% RSLogix 500 project LINCEBOT.RSS, saved by version 10.00.00.00 %
PROJECT "LINCEBOT"    % processor: MicroLogix 1400 %

PROGRAM FILES
  LAD 2   28 rungs
  LAD 4   10 rungs
  LAD 6   11 rungs
  LAD 8   6 rungs
  LAD 10   5 rungs
  LAD 12   10 rungs
  LAD 14   12 rungs
  LAD 16   4 rungs
  LAD 18   3 rungs
  LAD 20   3 rungs
  LAD 22   3 rungs
  LAD 24   13 rungs
  LAD 26   11 rungs
  LAD 80   9 rungs
  LAD 90   9 rungs
  LAD 100   27 rungs
  LAD 102   6 rungs
  LAD 103   6 rungs
  LAD 104   9 rungs
  LAD 105   8 rungs
  LAD 110   5 rungs
  LAD 111   8 rungs
  LAD 122   2 rungs
  LAD 125   7 rungs
  LAD 126   33 rungs
  LAD 131   2 rungs
  LAD 141   12 rungs
  LAD 150   11 rungs
  LAD 151   11 rungs
  LAD 160   42 rungs
  LAD 161   42 rungs
  LAD 170   10 rungs
  LAD 180   10 rungs
  LAD 70: only END

DATA FILES
  O0 OUTPUT  11 elements
  I1 INPUT  11 elements
  S2 STATUS  66 elements
  B3 BINARY  14 elements
  T4 TIMER  40 elements
  C5 COUNTER  1 elements
  R6 CONTROL  20 elements
  N7 INTEGER  200 elements
  F8 FLOAT  100 elements
  B9   256 elements
  B10   1 elements
  B11   256 elements
  B12   22 elements
  L13   100 elements
  F14   100 elements
  N15   100 elements
  L16   100 elements
  B17   128 elements
  B18   128 elements
  L23   100 elements
  L24   100 elements
  L42   52 elements
  B181   128 elements
  F182   50 elements
  L183   50 elements
  N184   50 elements
  B185   50 elements
  N186   50 elements
  L187   50 elements
  F188   50 elements
  B189   50 elements
  L190   50 elements
  B191   10 elements
  L192   50 elements
  F193   50 elements
  B194   128 elements
  B195   128 elements
  B196   50 elements
  N197   50 elements
  B198   50 elements
  L199   50 elements
  N200   50 elements
  L201   50 elements
  B202   50 elements
  N203   50 elements
  L204   50 elements
  F205   50 elements

LADDER 2
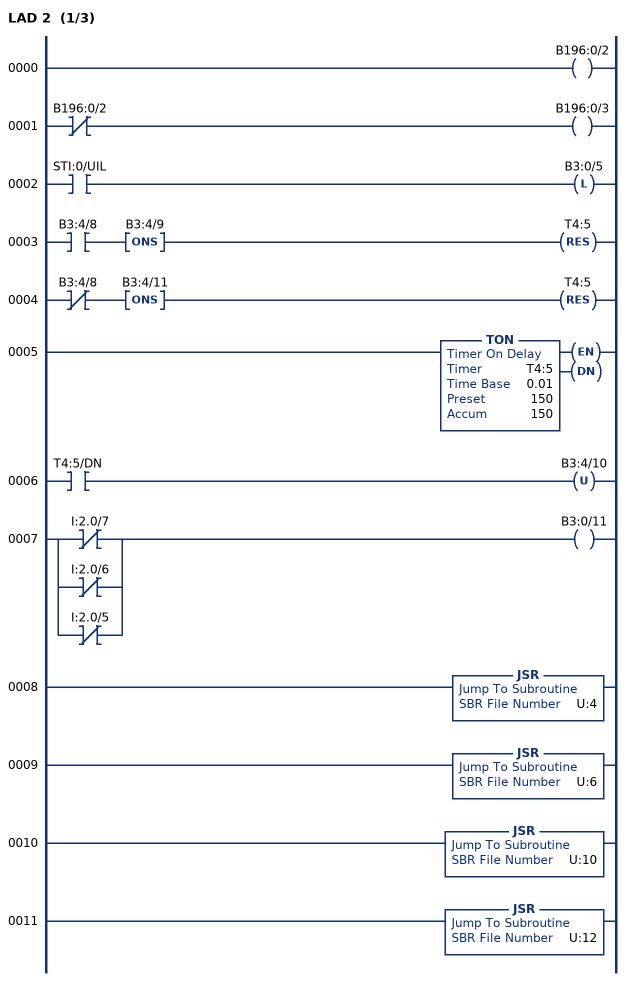
% Rung: 0 %
SOR OTE B196:0/2 EOR
% Rung: 1 %
SOR XIO B196:0/2 OTE B196:0/3 EOR
% Rung: 2 %
SOR XIC STI:0/UIL OTL B3:0/5 EOR
% Rung: 3 %
SOR XIC B3:4/8 ONS B3:4/9 RES T4:5 EOR
% Rung: 4 %
SOR XIO B3:4/8 ONS B3:4/11 RES T4:5 EOR
% Rung: 5 %
SOR TON T4:5 0.01 150 150 EOR
% Rung: 6 %
SOR XIC T4:5/DN OTU B3:4/10 EOR
% Rung: 7 %
SOR BST XIO I:2.0/7 NXB XIO I:2.0/6 NXB XIO I:2.0/5 BND OTE B3:0/11 EOR
% Rung: 8 %
SOR JSR U:4 EOR
% Rung: 9 %
SOR JSR U:6 EOR
% Rung: 10 %
SOR JSR U:10 EOR
% Rung: 11 %
SOR JSR U:12 EOR

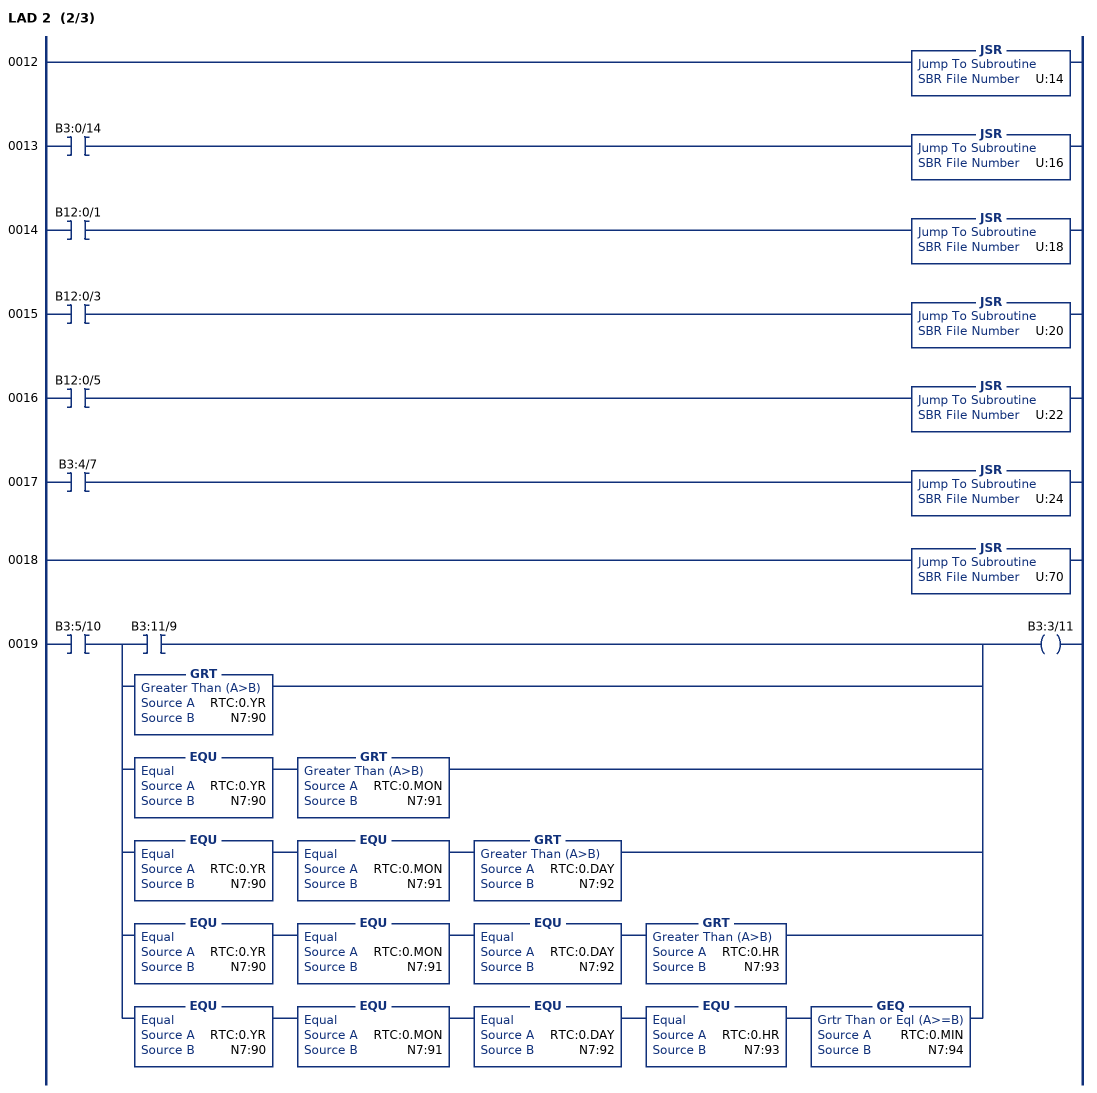
% Rung: 12 %
SOR JSR U:14 EOR
% Rung: 13 %
SOR XIC B3:0/14 JSR U:16 EOR
% Rung: 14 %
SOR XIC B12:0/1 JSR U:18 EOR
% Rung: 15 %
SOR XIC B12:0/3 JSR U:20 EOR
% Rung: 16 %
SOR XIC B12:0/5 JSR U:22 EOR
% Rung: 17 %
SOR XIC B3:4/7 JSR U:24 EOR
% Rung: 18 %
SOR JSR U:70 EOR
% Rung: 19 %
SOR XIC B3:5/10 BST XIC B3:11/9 NXB GRT RTC:0.YR N7:90 NXB EQU RTC:0.YR N7:90 GRT RTC:0.MON N7:91 NXB EQU RTC:0.YR N7:90 EQU RTC:0.MON N7:91 GRT RTC:0.DAY N7:92 NXB EQU RTC:0.YR N7:90 EQU RTC:0.MON N7:91 EQU RTC:0.DAY N7:92 GRT RTC:0.HR N7:93 NXB EQU RTC:0.YR N7:90 EQU RTC:0.MON N7:91 EQU RTC:0.DAY N7:92 EQU RTC:0.HR N7:93 GEQ RTC:0.MIN N7:94 BND OTE B3:3/11 EOR

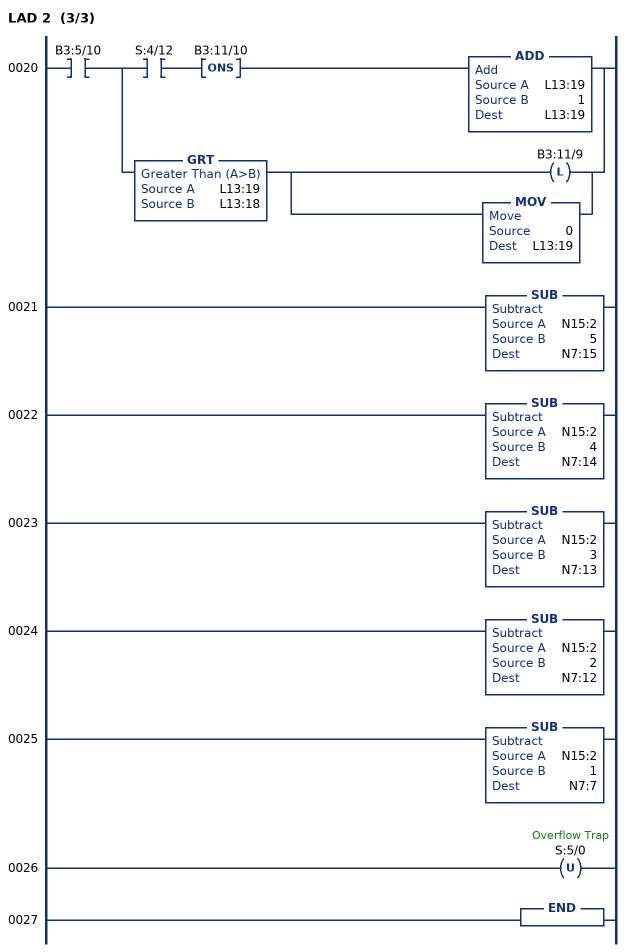
% Rung: 20 %
SOR XIC B3:5/10 BST XIC S:4/12 ONS B3:11/10 ADD L13:19 1 L13:19 NXB GRT L13:19 L13:18 BST OTL B3:11/9 NXB MOV 0 L13:19 BND BND EOR
% Rung: 21 %
SOR SUB N15:2 5 N7:15 EOR
% Rung: 22 %
SOR SUB N15:2 4 N7:14 EOR
% Rung: 23 %
SOR SUB N15:2 3 N7:13 EOR
% Rung: 24 %
SOR SUB N15:2 2 N7:12 EOR
% Rung: 25 %
SOR SUB N15:2 1 N7:7 EOR
% Rung: 26 %
SOR OTU S:5/0 EOR
%   S:5/0  "Overflow Trap" %
% Rung: 27 %
SOR END EOR

LADDER 4
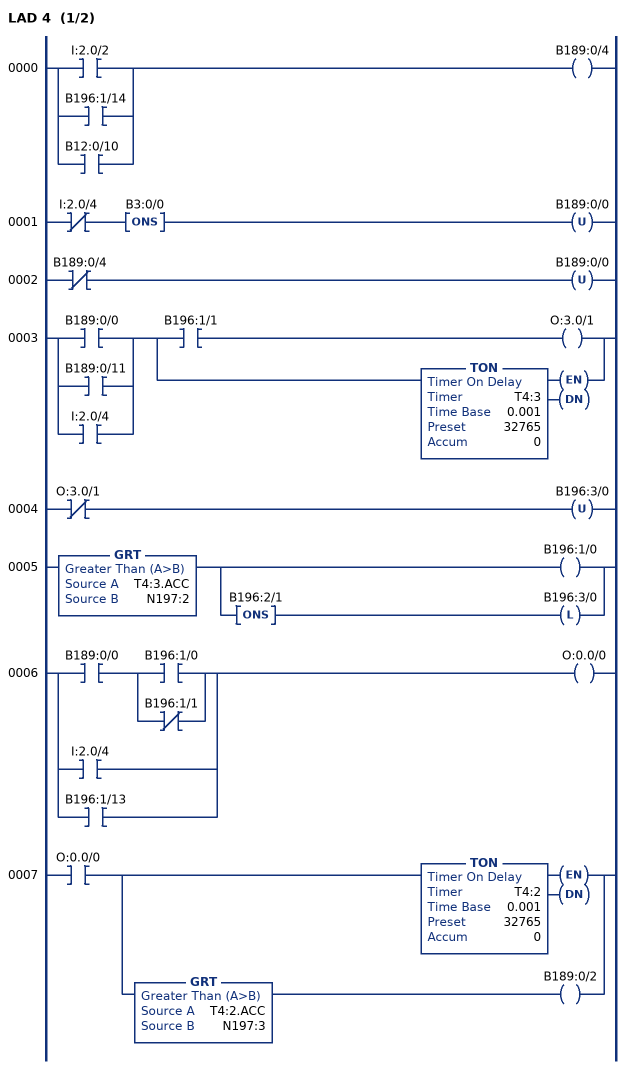
% Rung: 0 %
SOR BST XIC I:2.0/2 NXB XIC B196:1/14 NXB XIC B12:0/10 BND OTE B189:0/4 EOR
% Rung: 1 %
SOR XIO I:2.0/4 ONS B3:0/0 OTU B189:0/0 EOR
% Rung: 2 %
SOR XIO B189:0/4 OTU B189:0/0 EOR
% Rung: 3 %
SOR BST XIC B189:0/0 NXB XIC B189:0/11 NXB XIC I:2.0/4 BND BST XIC B196:1/1 OTE O:3.0/1 NXB TON T4:3 0.001 32765 0 BND EOR
% Rung: 4 %
SOR XIO O:3.0/1 OTU B196:3/0 EOR
% Rung: 5 %
SOR GRT T4:3.ACC N197:2 BST OTE B196:1/0 NXB ONS B196:2/1 OTL B196:3/0 BND EOR
% Rung: 6 %
SOR BST XIC B189:0/0 BST XIC B196:1/0 NXB XIO B196:1/1 BND NXB XIC I:2.0/4 NXB XIC B196:1/13 BND OTE O:0.0/0 EOR
% Rung: 7 %
SOR XIC O:0.0/0 BST TON T4:2 0.001 32765 0 NXB GRT T4:2.ACC N197:3 OTE B189:0/2 BND EOR

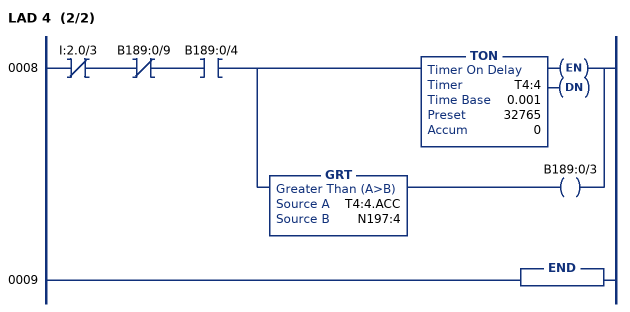
% Rung: 8 %
SOR XIO I:2.0/3 XIO B189:0/9 XIC B189:0/4 BST TON T4:4 0.001 32765 0 NXB GRT T4:4.ACC N197:4 OTE B189:0/3 BND EOR
% Rung: 9 %
SOR END EOR

LADDER 6
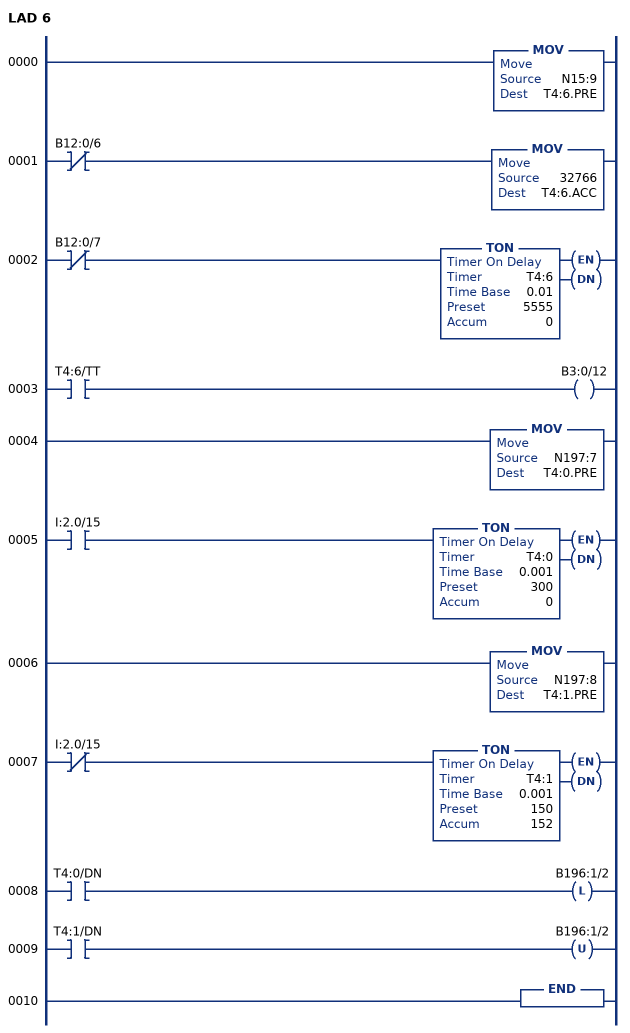
% Rung: 0 %
SOR MOV N15:9 T4:6.PRE EOR
% Rung: 1 %
SOR XIO B12:0/6 MOV 32766 T4:6.ACC EOR
% Rung: 2 %
SOR XIO B12:0/7 TON T4:6 0.01 5555 0 EOR
% Rung: 3 %
SOR XIC T4:6/TT OTE B3:0/12 EOR
% Rung: 4 %
SOR MOV N197:7 T4:0.PRE EOR
% Rung: 5 %
SOR XIC I:2.0/15 TON T4:0 0.001 300 0 EOR
% Rung: 6 %
SOR MOV N197:8 T4:1.PRE EOR
% Rung: 7 %
SOR XIO I:2.0/15 TON T4:1 0.001 150 152 EOR
% Rung: 8 %
SOR XIC T4:0/DN OTL B196:1/2 EOR
% Rung: 9 %
SOR XIC T4:1/DN OTU B196:1/2 EOR
% Rung: 10 %
SOR END EOR

LADDER 8
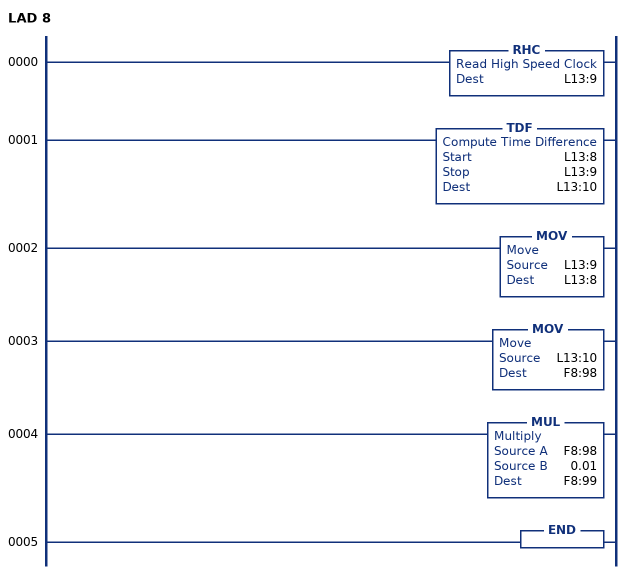
% Rung: 0 %
SOR RHC L13:9 EOR
% Rung: 1 %
SOR TDF L13:8 L13:9 L13:10 EOR
% Rung: 2 %
SOR MOV L13:9 L13:8 EOR
% Rung: 3 %
SOR MOV L13:10 F8:98 EOR
% Rung: 4 %
SOR MUL F8:98 0.01 F8:99 EOR
% Rung: 5 %
SOR END EOR

LADDER 10
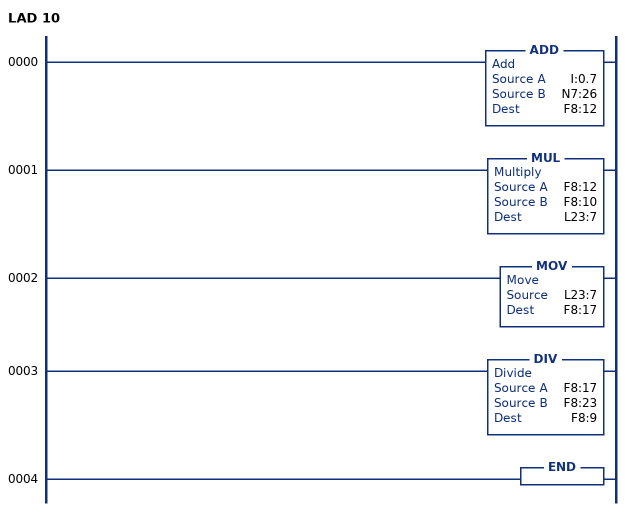
% Rung: 0 %
SOR ADD I:0.7 N7:26 F8:12 EOR
% Rung: 1 %
SOR MUL F8:12 F8:10 L23:7 EOR
% Rung: 2 %
SOR MOV L23:7 F8:17 EOR
% Rung: 3 %
SOR DIV F8:17 F8:23 F8:9 EOR
% Rung: 4 %
SOR END EOR

LADDER 12
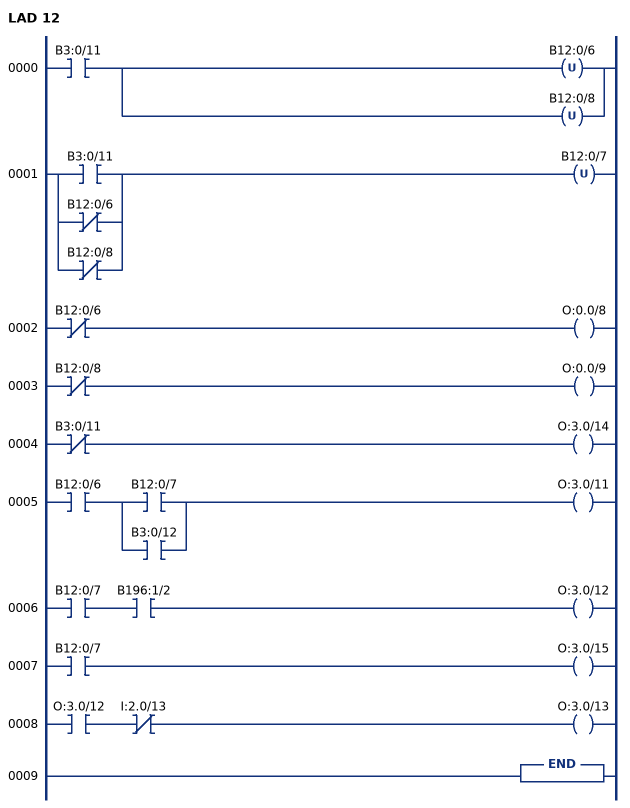
% Rung: 0 %
SOR XIC B3:0/11 BST OTU B12:0/6 NXB OTU B12:0/8 BND EOR
% Rung: 1 %
SOR BST XIC B3:0/11 NXB XIO B12:0/6 NXB XIO B12:0/8 BND OTU B12:0/7 EOR
% Rung: 2 %
SOR XIO B12:0/6 OTE O:0.0/8 EOR
% Rung: 3 %
SOR XIO B12:0/8 OTE O:0.0/9 EOR
% Rung: 4 %
SOR XIO B3:0/11 OTE O:3.0/14 EOR
% Rung: 5 %
SOR XIC B12:0/6 BST XIC B12:0/7 NXB XIC B3:0/12 BND OTE O:3.0/11 EOR
% Rung: 6 %
SOR XIC B12:0/7 XIC B196:1/2 OTE O:3.0/12 EOR
% Rung: 7 %
SOR XIC B12:0/7 OTE O:3.0/15 EOR
% Rung: 8 %
SOR XIC O:3.0/12 XIO I:2.0/13 OTE O:3.0/13 EOR
% Rung: 9 %
SOR END EOR

LADDER 14
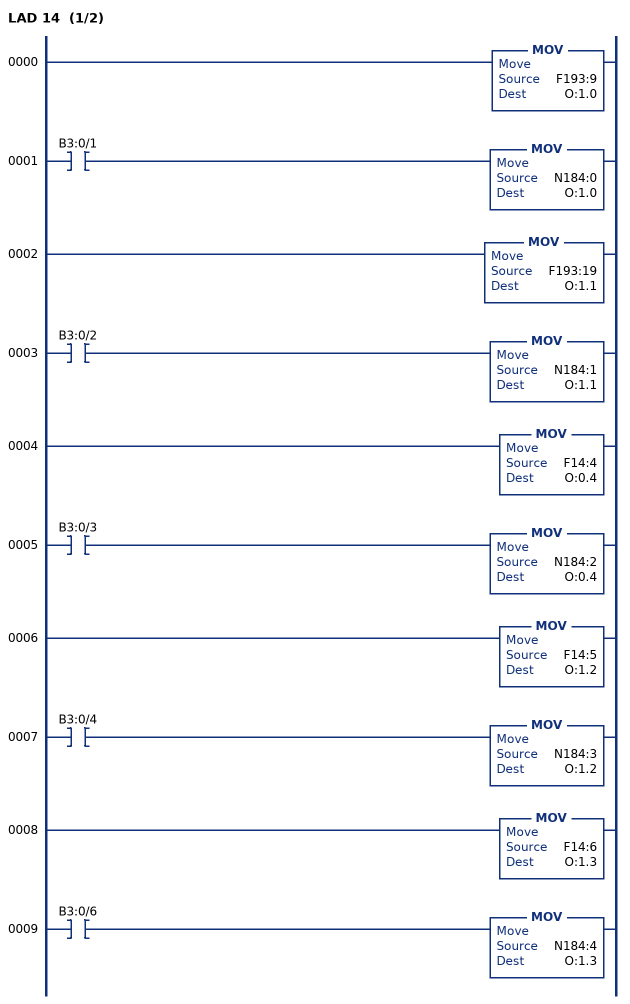
% Rung: 0 %
SOR MOV F193:9 O:1.0 EOR
% Rung: 1 %
SOR XIC B3:0/1 MOV N184:0 O:1.0 EOR
% Rung: 2 %
SOR MOV F193:19 O:1.1 EOR
% Rung: 3 %
SOR XIC B3:0/2 MOV N184:1 O:1.1 EOR
% Rung: 4 %
SOR MOV F14:4 O:0.4 EOR
% Rung: 5 %
SOR XIC B3:0/3 MOV N184:2 O:0.4 EOR
% Rung: 6 %
SOR MOV F14:5 O:1.2 EOR
% Rung: 7 %
SOR XIC B3:0/4 MOV N184:3 O:1.2 EOR
% Rung: 8 %
SOR MOV F14:6 O:1.3 EOR
% Rung: 9 %
SOR XIC B3:0/6 MOV N184:4 O:1.3 EOR

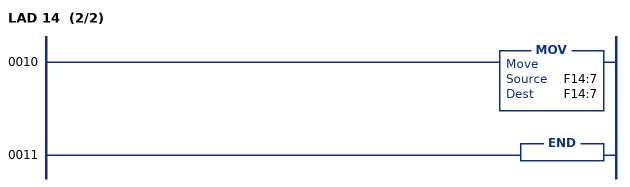
% Rung: 10 %
SOR MOV F14:7 F14:7 EOR
% Rung: 11 %
SOR END EOR

LADDER 16
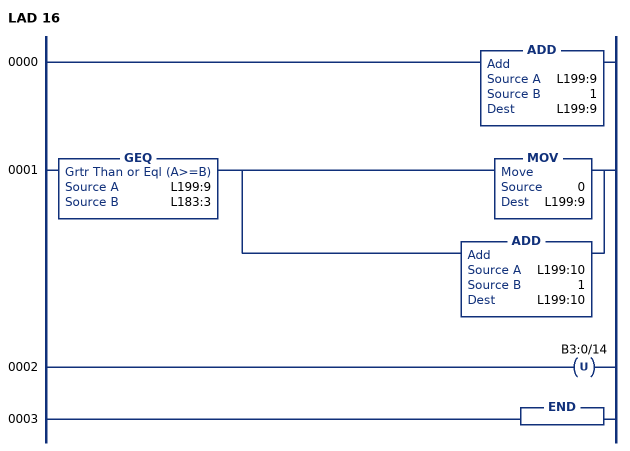
% Rung: 0 %
SOR ADD L199:9 1 L199:9 EOR
% Rung: 1 %
SOR GEQ L199:9 L183:3 BST MOV 0 L199:9 NXB ADD L199:10 1 L199:10 BND EOR
% Rung: 2 %
SOR OTU B3:0/14 EOR
% Rung: 3 %
SOR END EOR

LADDER 18
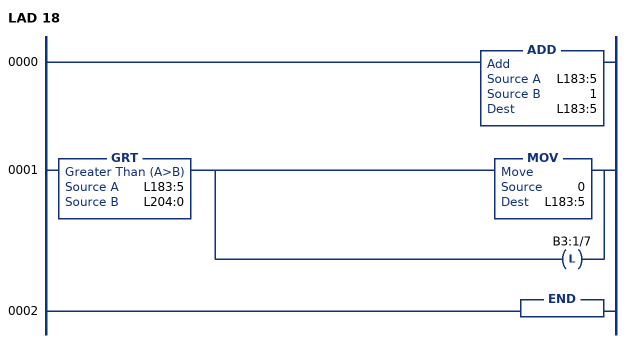
% Rung: 0 %
SOR ADD L183:5 1 L183:5 EOR
% Rung: 1 %
SOR GRT L183:5 L204:0 BST MOV 0 L183:5 NXB OTL B3:1/7 BND EOR
% Rung: 2 %
SOR END EOR

LADDER 20
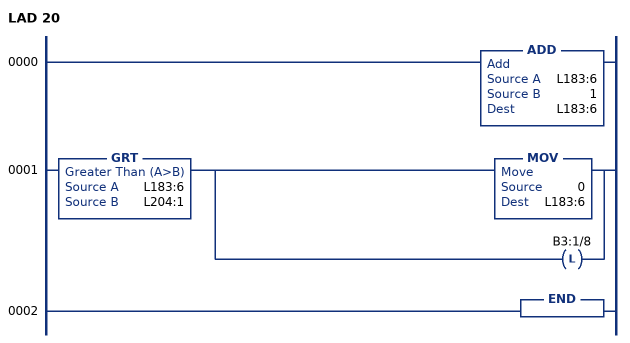
% Rung: 0 %
SOR ADD L183:6 1 L183:6 EOR
% Rung: 1 %
SOR GRT L183:6 L204:1 BST MOV 0 L183:6 NXB OTL B3:1/8 BND EOR
% Rung: 2 %
SOR END EOR

LADDER 22
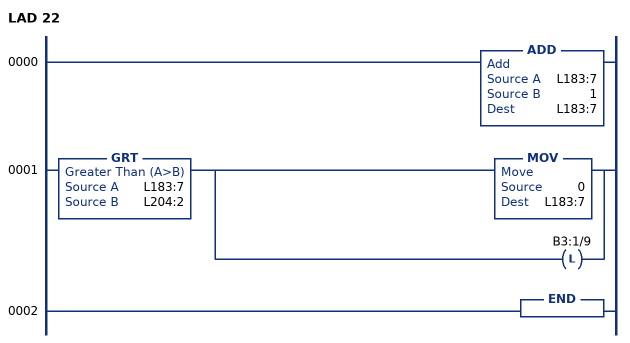
% Rung: 0 %
SOR ADD L183:7 1 L183:7 EOR
% Rung: 1 %
SOR GRT L183:7 L204:2 BST MOV 0 L183:7 NXB OTL B3:1/9 BND EOR
% Rung: 2 %
SOR END EOR

LADDER 24
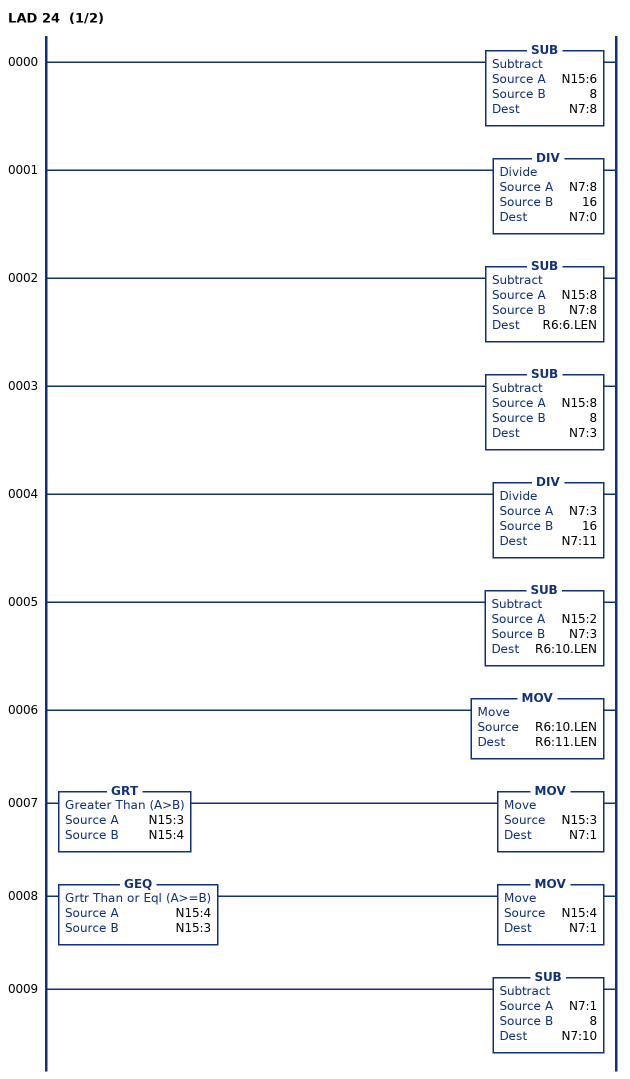
% Rung: 0 %
SOR SUB N15:6 8 N7:8 EOR
% Rung: 1 %
SOR DIV N7:8 16 N7:0 EOR
% Rung: 2 %
SOR SUB N15:8 N7:8 R6:6.LEN EOR
% Rung: 3 %
SOR SUB N15:8 8 N7:3 EOR
% Rung: 4 %
SOR DIV N7:3 16 N7:11 EOR
% Rung: 5 %
SOR SUB N15:2 N7:3 R6:10.LEN EOR
% Rung: 6 %
SOR MOV R6:10.LEN R6:11.LEN EOR
% Rung: 7 %
SOR GRT N15:3 N15:4 MOV N15:3 N7:1 EOR
% Rung: 8 %
SOR GEQ N15:4 N15:3 MOV N15:4 N7:1 EOR
% Rung: 9 %
SOR SUB N7:1 8 N7:10 EOR

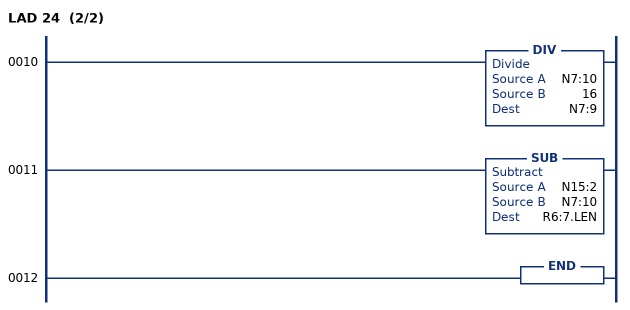
% Rung: 10 %
SOR DIV N7:10 16 N7:9 EOR
% Rung: 11 %
SOR SUB N15:2 N7:10 R6:7.LEN EOR
% Rung: 12 %
SOR END EOR

LADDER 26
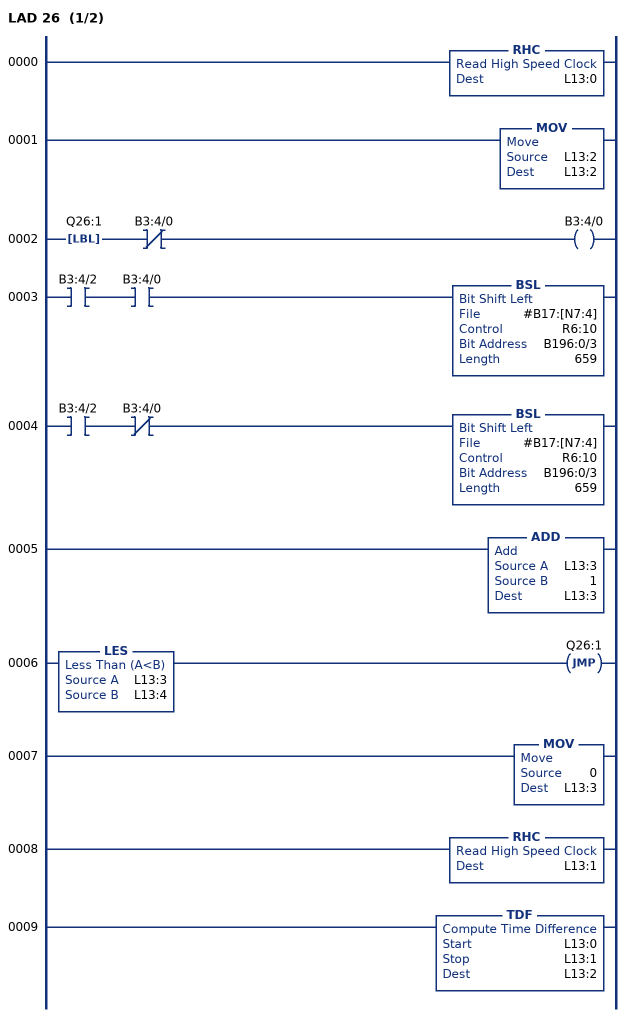
% Rung: 0 %
SOR RHC L13:0 EOR
% Rung: 1 %
SOR MOV L13:2 L13:2 EOR
% Rung: 2 %
SOR LBL Q26:1 XIO B3:4/0 OTE B3:4/0 EOR
% Rung: 3 %
SOR XIC B3:4/2 XIC B3:4/0 BSL #B17:[N7:4] R6:10 B196:0/3 659 EOR
% Rung: 4 %
SOR XIC B3:4/2 XIO B3:4/0 BSL #B17:[N7:4] R6:10 B196:0/3 659 EOR
% Rung: 5 %
SOR ADD L13:3 1 L13:3 EOR
% Rung: 6 %
SOR LES L13:3 L13:4 JMP Q26:1 EOR
% Rung: 7 %
SOR MOV 0 L13:3 EOR
% Rung: 8 %
SOR RHC L13:1 EOR
% Rung: 9 %
SOR TDF L13:0 L13:1 L13:2 EOR

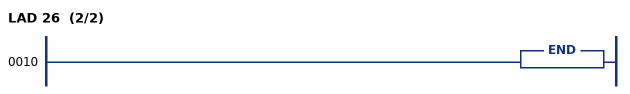
% Rung: 10 %
SOR END EOR

LADDER 80
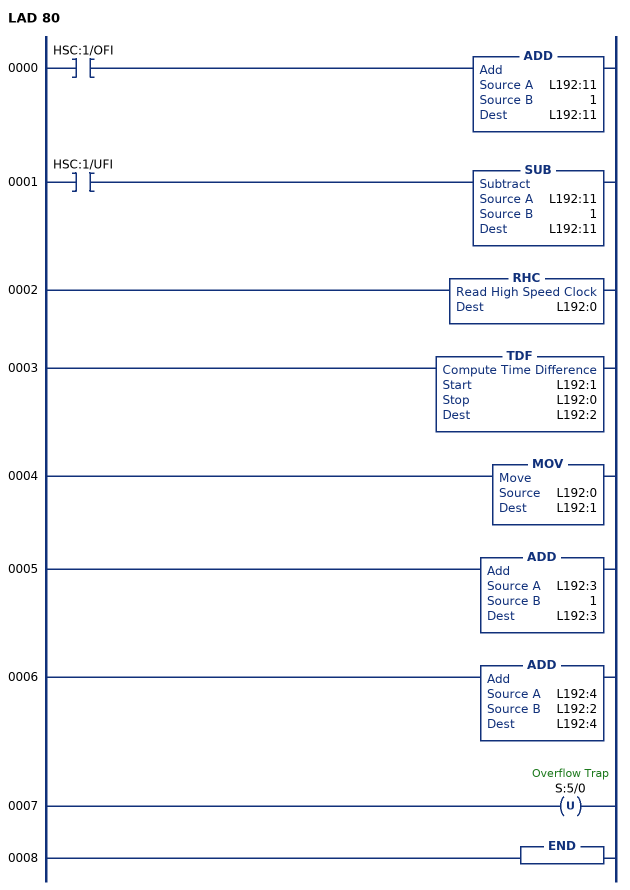
% Rung: 0 %
SOR XIC HSC:1/OFI ADD L192:11 1 L192:11 EOR
% Rung: 1 %
SOR XIC HSC:1/UFI SUB L192:11 1 L192:11 EOR
% Rung: 2 %
SOR RHC L192:0 EOR
% Rung: 3 %
SOR TDF L192:1 L192:0 L192:2 EOR
% Rung: 4 %
SOR MOV L192:0 L192:1 EOR
% Rung: 5 %
SOR ADD L192:3 1 L192:3 EOR
% Rung: 6 %
SOR ADD L192:4 L192:2 L192:4 EOR
% Rung: 7 %
SOR OTU S:5/0 EOR
%   S:5/0  "Overflow Trap" %
% Rung: 8 %
SOR END EOR

LADDER 90
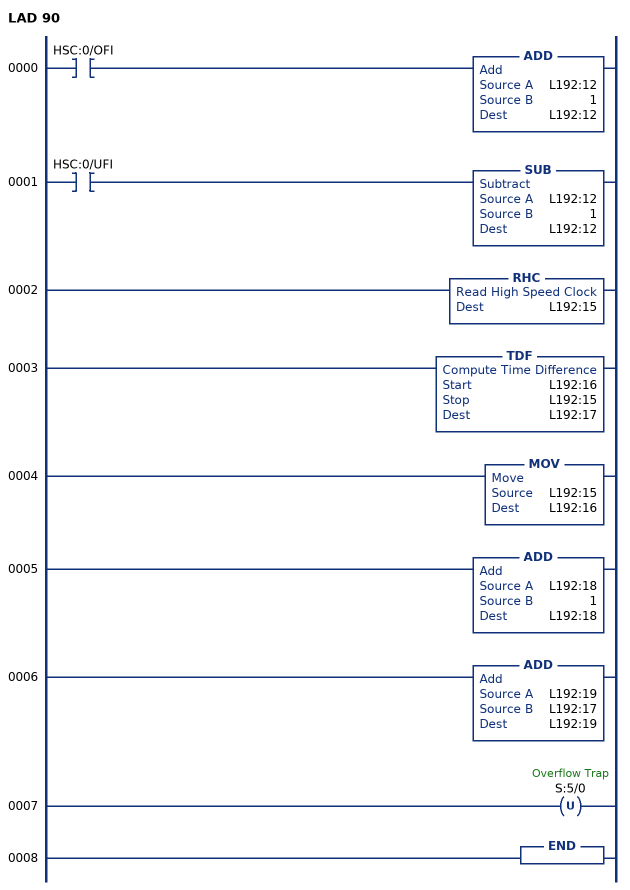
% Rung: 0 %
SOR XIC HSC:0/OFI ADD L192:12 1 L192:12 EOR
% Rung: 1 %
SOR XIC HSC:0/UFI SUB L192:12 1 L192:12 EOR
% Rung: 2 %
SOR RHC L192:15 EOR
% Rung: 3 %
SOR TDF L192:16 L192:15 L192:17 EOR
% Rung: 4 %
SOR MOV L192:15 L192:16 EOR
% Rung: 5 %
SOR ADD L192:18 1 L192:18 EOR
% Rung: 6 %
SOR ADD L192:19 L192:17 L192:19 EOR
% Rung: 7 %
SOR OTU S:5/0 EOR
%   S:5/0  "Overflow Trap" %
% Rung: 8 %
SOR END EOR

LADDER 100
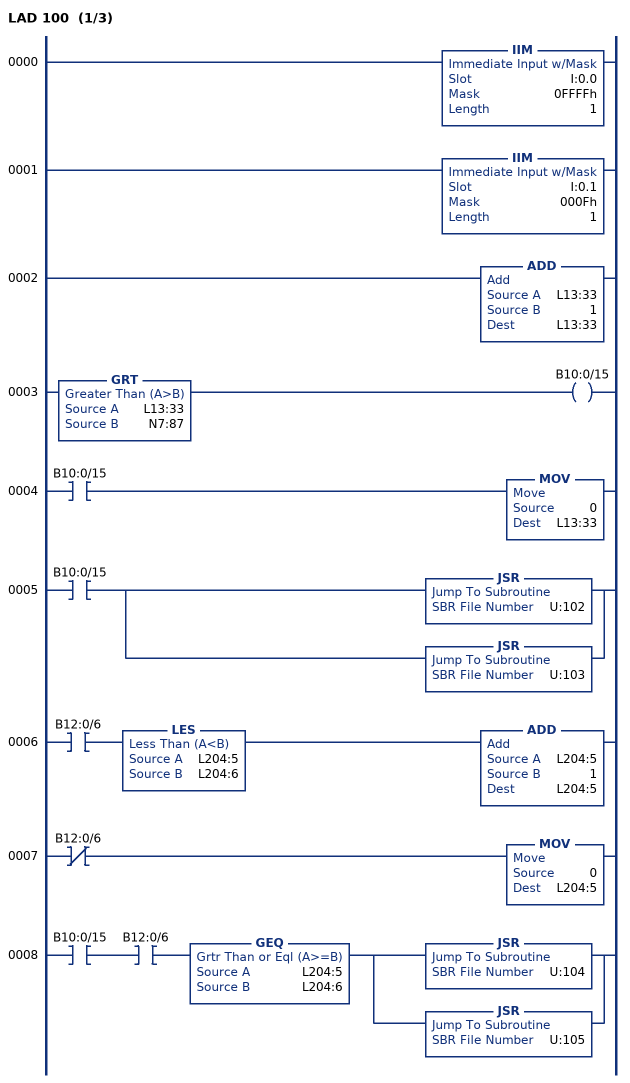
% Rung: 0 %
SOR IIM I:0.0 0FFFFh 1 EOR
% Rung: 1 %
SOR IIM I:0.1 000Fh 1 EOR
% Rung: 2 %
SOR ADD L13:33 1 L13:33 EOR
% Rung: 3 %
SOR GRT L13:33 N7:87 OTE B10:0/15 EOR
% Rung: 4 %
SOR XIC B10:0/15 MOV 0 L13:33 EOR
% Rung: 5 %
SOR XIC B10:0/15 BST JSR U:102 NXB JSR U:103 BND EOR
% Rung: 6 %
SOR XIC B12:0/6 LES L204:5 L204:6 ADD L204:5 1 L204:5 EOR
% Rung: 7 %
SOR XIO B12:0/6 MOV 0 L204:5 EOR
% Rung: 8 %
SOR XIC B10:0/15 XIC B12:0/6 GEQ L204:5 L204:6 BST JSR U:104 NXB JSR U:105 BND EOR

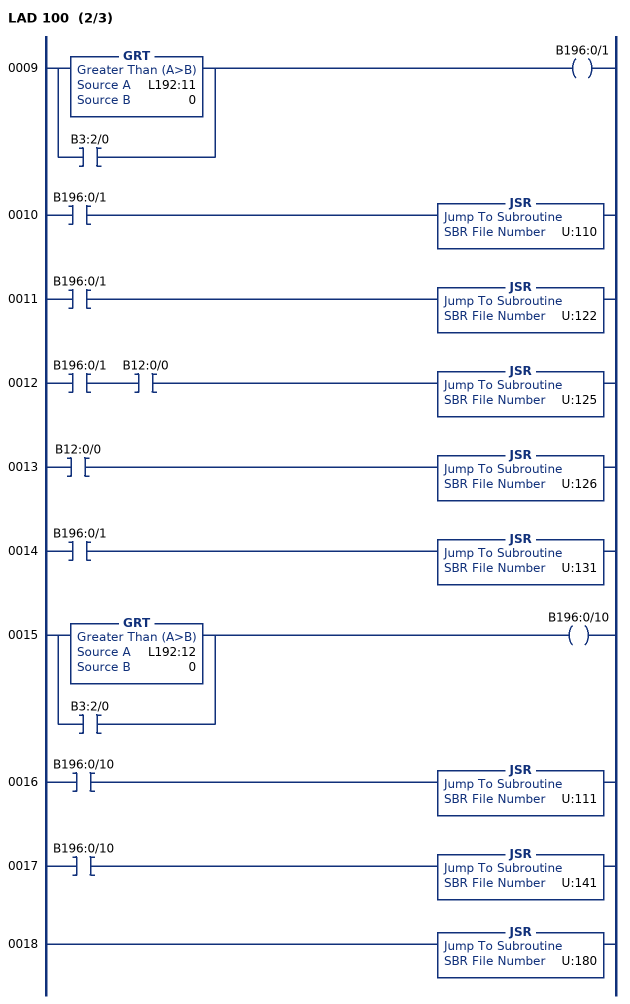
% Rung: 9 %
SOR BST GRT L192:11 0 NXB XIC B3:2/0 BND OTE B196:0/1 EOR
% Rung: 10 %
SOR XIC B196:0/1 JSR U:110 EOR
% Rung: 11 %
SOR XIC B196:0/1 JSR U:122 EOR
% Rung: 12 %
SOR XIC B196:0/1 XIC B12:0/0 JSR U:125 EOR
% Rung: 13 %
SOR XIC B12:0/0 JSR U:126 EOR
% Rung: 14 %
SOR XIC B196:0/1 JSR U:131 EOR
% Rung: 15 %
SOR BST GRT L192:12 0 NXB XIC B3:2/0 BND OTE B196:0/10 EOR
% Rung: 16 %
SOR XIC B196:0/10 JSR U:111 EOR
% Rung: 17 %
SOR XIC B196:0/10 JSR U:141 EOR
% Rung: 18 %
SOR JSR U:180 EOR

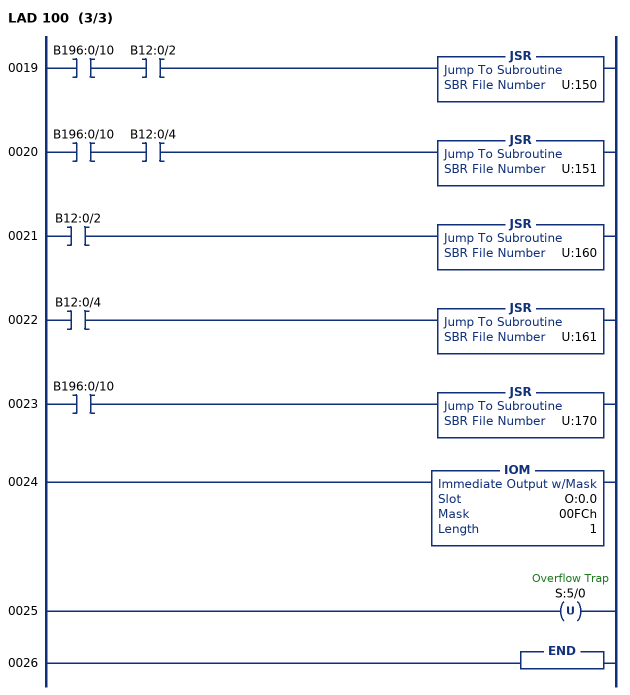
% Rung: 19 %
SOR XIC B196:0/10 XIC B12:0/2 JSR U:150 EOR
% Rung: 20 %
SOR XIC B196:0/10 XIC B12:0/4 JSR U:151 EOR
% Rung: 21 %
SOR XIC B12:0/2 JSR U:160 EOR
% Rung: 22 %
SOR XIC B12:0/4 JSR U:161 EOR
% Rung: 23 %
SOR XIC B196:0/10 JSR U:170 EOR
% Rung: 24 %
SOR IOM O:0.0 00FCh 1 EOR
% Rung: 25 %
SOR OTU S:5/0 EOR
%   S:5/0  "Overflow Trap" %
% Rung: 26 %
SOR END EOR

LADDER 102
